// TIA Portal V17 export
// export: Created 2022-06-27T13:56:11.0548451Z, ExportSetting WithDefaults, DisplayName Totally Integrated Automation Portal, DisplayVersion V17 Update 3, DisplayName TIA Portal Openness, DisplayVersion V17 Update 3, DisplayName TIA Portal Version Control Interface, DisplayVersion V17, DisplayName SINAMICS Startdrive Advanced, DisplayVersion V17 Update1, DisplayName SINAMICS Startdrive G110M, G120, G120C, G120D, G120P, G115D, DisplayVersion V17 Update1, DisplayName SINAMICS Startdrive G130, G150, S120, S150, SINAMICS MV, S210, DisplayVersion V17 Update1, DisplayName STEP 7 Professional, DisplayVersion V17 Update 3, DisplayName STEP 7 Safety, DisplayVersion V17, DisplayName WinCC UA Professional, DisplayVersion V17 Update 3
FUNCTION_BLOCK "S02_CTRL_TURBO"   // FB2, LAD
{ S7_Optimized_Access := 'TRUE' }
VERSION : 0.1
// stored: AutoNumber false, IsIECCheckEnabled false, IsRetainMemResEnabled false, MemoryReserve 100, SetENOAutomatically false, UDAEnableTagReadback false
BEGIN

REGION Network 1: Calls all subfunctions
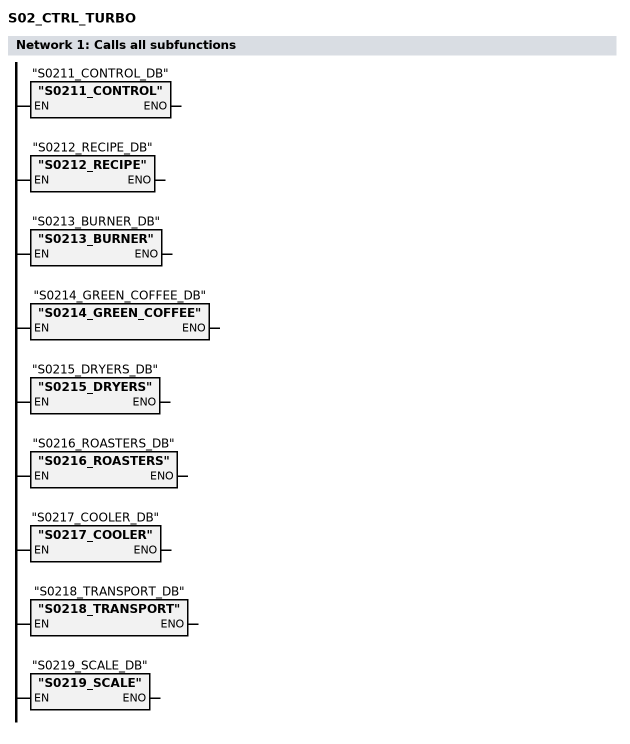
   RUNG wire#powerrail
      "S0211_CONTROL_DB"()
   END_RUNG
   RUNG wire#powerrail
      "S0212_RECIPE_DB"()
   END_RUNG
   RUNG wire#powerrail
      "S0213_BURNER_DB"()
   END_RUNG
   RUNG wire#powerrail
      "S0214_GREEN_COFFEE_DB"()
   END_RUNG
   RUNG wire#powerrail
      "S0215_DRYERS_DB"()
   END_RUNG
   RUNG wire#powerrail
      "S0216_ROASTERS_DB"()
   END_RUNG
   RUNG wire#powerrail
      "S0217_COOLER_DB"()
   END_RUNG
   RUNG wire#powerrail
      "S0218_TRANSPORT_DB"()
   END_RUNG
   RUNG wire#powerrail
      "S0219_SCALE_DB"()
   END_RUNG
   // the same network as SCL:
   "S0211_CONTROL_DB"();   // "S0211_CONTROL"
   "S0212_RECIPE_DB"();   // "S0212_RECIPE"
   "S0213_BURNER_DB"();   // "S0213_BURNER"
   "S0214_GREEN_COFFEE_DB"();   // "S0214_GREEN_COFFEE"
   "S0215_DRYERS_DB"();   // "S0215_DRYERS"
   "S0216_ROASTERS_DB"();   // "S0216_ROASTERS"
   "S0217_COOLER_DB"();   // "S0217_COOLER"
   "S0218_TRANSPORT_DB"();   // "S0218_TRANSPORT"
   "S0219_SCALE_DB"();   // "S0219_SCALE"
END_REGION
END_FUNCTION_BLOCK
